FUNCTION FC_CalculateYCenterPoint : REAL		// Calculates the center point (Y) of 2 points
VAR_INPUT
	iPoint1:		TcVnPoint2_REAL;
	iPoint2:		TcVnPoint2_REAL;
END_VAR

FC_CalculateYCenterPoint := (iPoint1[VISION.Y_COORD] + iPoint2[VISION.Y_COORD]) / 2;

END_FUNCTION

(* stored: Version 1.1.0.1
   POU FC_CalculateYCenterPoint: Id {49ce58a3-3206-436e-97aa-da292a8929cc}, SpecialFunc None *)
